// Mitsubishi GX Works2 project: Vacuum ST Code   PLC: FX1S

// global labels: Global1
VAR_GLOBAL
  runAutoFlag : BOOL;
  conveyorRunFlag : BOOL;
  solenoidRunFlag : BOOL;
  vacuumRunFlag : BOOL;
  runAutoStatus : INT;
  btnStart AT X000 : BOOL;
  btnStop AT X001 : BOOL;
  senProximity AT X002 : BOOL;
  rConveyor AT Y002 : BOOL;
  rSolenoid AT Y001 : BOOL;
  rVacuumStart AT Y000 : BOOL;
  clickVacuumRunFlag : BOOL;
END_VAR
VAR_GLOBAL CONSTANT
  tClickStartVacuum : TIME := T#1s;
  tVacuum : TIME := T#50s;
  tAfterVacuum : TIME := T#3s;
  tAfterVacuumConveyor : TIME := T#15s;
  tValidateSensor : TIME := T#3s;
  tSolenoidClose : TIME := T#2s;
END_VAR
VAR_GLOBAL
  rLightConveyor AT Y005 : BOOL;
  rLightSolenoid AT Y007 : BOOL;
  rLightClick AT Y006 : BOOL;
  rLightSensor AT Y010 : BOOL;
  rLightStart AT Y003 : BOOL;
  rLightStop AT Y004 : BOOL;
  btnManConveyor AT X003 : BOOL;
  btnManSolenoid AT X004 : BOOL;
  btnManClickVacuum AT X005 : BOOL;
  ManRunFlagConveyor : BOOL;
  ManRunFlagSolenoid : BOOL;
  ManRunFlagClickVacuum : BOOL;
END_VAR

// task Task_01 (event TRUE, interval 0, priority 31): POU_01

PROGRAM POU_01
VAR
  Conveyor : RunOutput;
  Solenoid : RunOutput;
  ClickStartVaccum : RunOutput;
  EValidateTimer : TIME;
  ValidateTimer : TON;
  CloseSolenoidTimer : TON;
  ECloseSolenoidTimer : TIME;
  ClickStartTimer : TON;
  EClickStartTimer : TIME;
  VacuumTimer : TON;
  EVacuumTimer : TIME;
  AfterVacuumTimer : TON;
  EAfterVacuumTimer : TIME;
  AfterVacuumConveyorTimer : TON;
  EAfterVacuumConveyorTimer : TIME;
  ManualRunConveyor : RunOutput;
  ManualRunSolenoid : RunOutput;
  ManualRunClickVacuum : RunOutput;
  LightRunStart : RunOutput;
  LightRunStop : RunOutput;
  LightRunConveyor : RunOutput;
  LightRunSolenoid : RunOutput;
  LightRunClickVacuum : RunOutput;
  LightRunSensor : RunOutput;
  ConveyorManualRun : RunOutput;
  ConveyorManualRunOnOff : StartStop;
  SolenoidManualRunOnOff : StartStop;
  ClickVacuumManualRunOnOff : StartStop;
END_VAR
(* Start Run Auto *)
IF	btnStart = TRUE THEN
	runAutoFlag := TRUE;
	runAutoStatus := 1;
END_IF;

(* Stop Alll *)
IF btnStop = TRUE THEN
	runAutoFlag := FALSE;
	conveyorRunFlag:= FALSE;
	solenoidRunFlag:= FALSE;
	clickVacuumRunFlag := FALSE;
	rConveyor := FALSE;
	rSolenoid := FALSE;
	rVacuumStart := FALSE;
	runAutoStatus := 0;
END_IF;

(* Run Auto Sequence *)
IF runAutoFlag  = 1 THEN
	CASE runAutoStatus OF
		1:
		(* RUN CONVEYOR AND WAIT FOR THE SENSOR TO SENSE*)
			IF senProximity = TRUE THEN
				conveyorRunFlag:= FALSE;
				runAutoStatus := 2;
			ELSE
				conveyorRunFlag:= TRUE;
			END_IF;
		2:
		(* VALIDATE SENSOR INPUT*)
			IF senProximity = TRUE THEN
				ValidateTimer(IN:= TRUE ,PT:= tValidateSensor , ET:=EValidateTimer);
				IF ValidateTimer.Q = TRUE THEN
					ValidateTimer(IN:=FALSE);
					runAutoStatus := 3; 
				END_IF;
			ELSE
				ValidateTimer(IN:=FALSE);
				runAutoStatus := 1;
			END_IF;
		3:
		(* CLOSE SOLENOID *)
		CloseSolenoidTimer(IN:= TRUE ,PT:= tSolenoidClose, ET:= ECloseSolenoidTimer);
			IF CloseSolenoidTimer.Q = TRUE THEN
				CloseSolenoidTimer(IN:=FALSE);
				runAutoStatus := 4;
			ELSE
				 solenoidRunFlag:= TRUE;
			END_IF;
		4:
		(* RUN CLICK THE VACUUM START *)
			ClickStartTimer(IN:= TRUE ,PT:= tClickStartVacuum, ET:= EClickStartTimer);
			IF ClickStartTimer.Q = TRUE THEN
				ClickStartTimer(IN:=FALSE);
				clickVacuumRunFlag := FALSE;
				runAutoStatus := 5;
			ELSE
				 clickVacuumRunFlag := TRUE;
			END_IF;
		5:
		(* RUN VACUUM TIMER *)
			VacuumTimer(IN:= TRUE ,PT:= tVacuum, ET:= EVacuumTimer);
			IF VacuumTimer.Q = TRUE THEN
				VacuumTimer(IN:=FALSE);
				runAutoStatus := 6;
			END_IF;
		6:
		(* RUN VACUUM DELAY TIMER *)
			AfterVacuumTimer(IN:= TRUE ,PT:= tAfterVacuum, ET:= EAfterVacuumTimer);
			IF AfterVacuumTimer.Q = TRUE THEN
				AfterVacuumTimer(IN:=FALSE);
				runAutoStatus := 7;
			ELSE
				solenoidRunFlag := FALSE;
			END_IF;
		7:
		(* RUN VACUUM DELAY CONVEYOR ON TIMER *)
			AfterVacuumConveyorTimer(IN:= TRUE ,PT:= tAfterVacuumConveyor, ET:= EAfterVacuumConveyorTimer);
			IF AfterVacuumConveyorTimer.Q = TRUE THEN
				runAutoStatus := 1;
				AfterVacuumConveyorTimer(IN:=FALSE);
			ELSE
				conveyorRunFlag:= TRUE;
			END_IF;
	END_CASE;
ELSE
	(* Manual Run Conveyor *)
	IF ManRunFlagSolenoid = FALSE THEN
		ConveyorManualRunOnOff(btnInput:= btnManConveyor ,memoryOn:= M1 ,memoryOff:= M2 ,memoryOutput:= ManRunFlagConveyor );
	END_IF;
	
	IF ManRunFlagConveyor = FALSE THEN
		SolenoidManualRunOnOff(btnInput:= btnManSolenoid,memoryOn:= M3 ,memoryOff:= M4 ,memoryOutput:= ManRunFlagSolenoid);
	END_IF;
	
	IF ManRunFlagSolenoid = TRUE THEN
		ClickVacuumManualRunOnOff(btnInput:= btnManClickVacuum ,memoryOn:= M5 ,memoryOff:= M6,memoryOutput:= ManRunFlagClickVacuum);
	END_IF;
END_IF;

(* RUN MOTORS *)
IF runAutoFlag = TRUE THEN
	Conveyor(input := conveyorRunFlag ,output := rConveyor );
	Solenoid(input:= solenoidRunFlag ,output:= rSolenoid );
	ClickStartVaccum(input:= clickVacuumRunFlag ,output:= rVacuumStart );
ELSE
	ManualRunConveyor(input:= ManRunFlagConveyor ,output:= rConveyor  );
	ManualRunSolenoid(input:= ManRunFlagSolenoid ,output:= rSolenoid );
	ManualRunClickVacuum(input:= ManRunFlagClickVacuum ,output:= rVacuumStart  );
END_IF;
LightRunStart(input:= runAutoFlag ,output:= rLightStart );
LightRunStop(input:= NOT runAutoFlag ,output:= rLightStop );
LightRunConveyor(input:= rConveyor ,output:= rLightConveyor );
LightRunSolenoid(input:= rSolenoid ,output:= rLightSolenoid );
LightRunClickVacuum(input:= rVacuumStart ,output:= rLightClick );
LightRunSensor(input:= senProximity ,output:= rLightSensor);
END_PROGRAM

FUNCTION_BLOCK RunOutput
VAR_INPUT
  input : BOOL;
END_VAR
VAR_OUTPUT
  output : BOOL;
END_VAR
(* structured ladder/FBD written out as ST: instructions are called as NAME(EN, inputs, outputs); _pN, _eN, _tN stand for wires *)
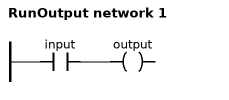
(* network 1 *)
output := input;
END_FUNCTION_BLOCK

FUNCTION_BLOCK StartStop
VAR_INPUT
  btnInput : BOOL;
END_VAR
VAR_IN_OUT
  memoryOn : BOOL;
  memoryOff : BOOL;
END_VAR
VAR_OUTPUT
  memoryOutput : BOOL;
END_VAR
(* structured ladder/FBD written out as ST: instructions are called as NAME(EN, inputs, outputs); _pN, _eN, _tN stand for wires *)
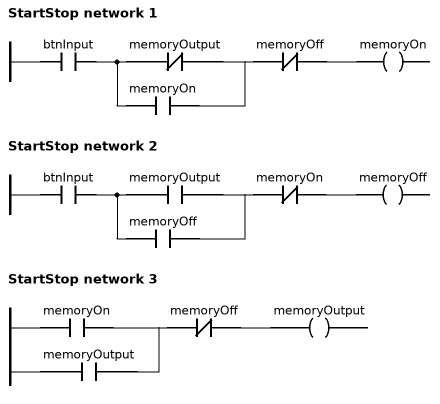
(* network 1 *)
memoryOn := ((btnInput AND NOT memoryOutput) OR (btnInput AND memoryOn)) AND NOT memoryOff;
(* network 2 *)
memoryOff := ((btnInput AND memoryOutput) OR (btnInput AND memoryOff)) AND NOT memoryOn;
(* network 3 *)
memoryOutput := (memoryOn OR memoryOutput) AND NOT memoryOff;
END_FUNCTION_BLOCK
